{attribute addProperty BoxType "BK1150-0000-0016"}
{attribute addProperty Id "Term_383_KL1002KL1002_D229A9CA00"}
{attribute addProperty CRC "2132326926"}
{attribute addProperty SizeInBites "0"}
{attribute addProperty SizeInBytes "0"}
TYPE A_0010_BK1150_0000_0016_7F18BA0E EXTENDS BK1150_4487A81F :
STRUCT
	{attribute addProperty Name "Term_383_KL1002"}
	Term_383_KL1002 : KL1002_D229A9CA;
END_STRUCT
END_TYPE

(* stored: Version 1.2.0.0, ProductVersion 3.1.4024.9
   DUT A_0010_BK1150_0000_0016_7F18BA0E: Id {c904b34a-4e97-4003-834d-72aaeeadba51} *)
